(* PLC project Scenario13_Final.project, CODESYS CODESYS V3.5 SP4 Patch 4 *)
(* stored: creationDateTime 2014-06-27T19:19:34.1584235, modificationDateTime 2014-06-20T17:27:16 *)

FUNCTION_BLOCK Crane
  VAR_INPUT
    SliderNotMovedOut : BOOL;
    SliderMovedOut : BOOL;
    MagazinCapacitiveSensor : BOOL;
    WorkpieceReady : BOOL;
    CraneDown : BOOL;
    CraneUp : BOOL;
    CraneSucked : BOOL;  (* CraneOnConveyor : BOOL; CraneOnMagazin : BOOL; *)
    StampLowered : BOOL;
    MagazinOpticalSensor : BOOL;  (* CranePositionStamp : BOOL; *)
    StampSliderFilled : BOOL;
    AnalogCranePosition : INT;
    StartButtonMagazin : BOOL;
    SFCReset : BOOL;
    StartVar : BOOL;
    StampSliderSensorMovedOut : BOOL;
  END_VAR
  VAR_OUTPUT
    CraneLower : BOOL;
    MagazinVacuumOff : BOOL;
    MagazinVacuumOn : BOOL;
    CraneTurnCounterclockwise : BOOL;
    CraneTurnClockwise : BOOL;
    MagazinSlider : BOOL;
    AnalogCranePressure : INT;
    StartCommandCrane : BOOL;
  END_VAR
  VAR
    Timer1 : TON;
    Duration1 : TIME := TIME#1s500ms;
    actualtime1 : TIME;
    interconnect : BOOL;
    interconnectCraneStartCommand : BOOL;
    TimeDelay_Timer : TON;
    TimeDelay_Timer_Duration : TIME := TIME#50ms;
    TimeDelay_Timer_interconnect : BOOL;
    SFCInit : BOOL;
  END_VAR

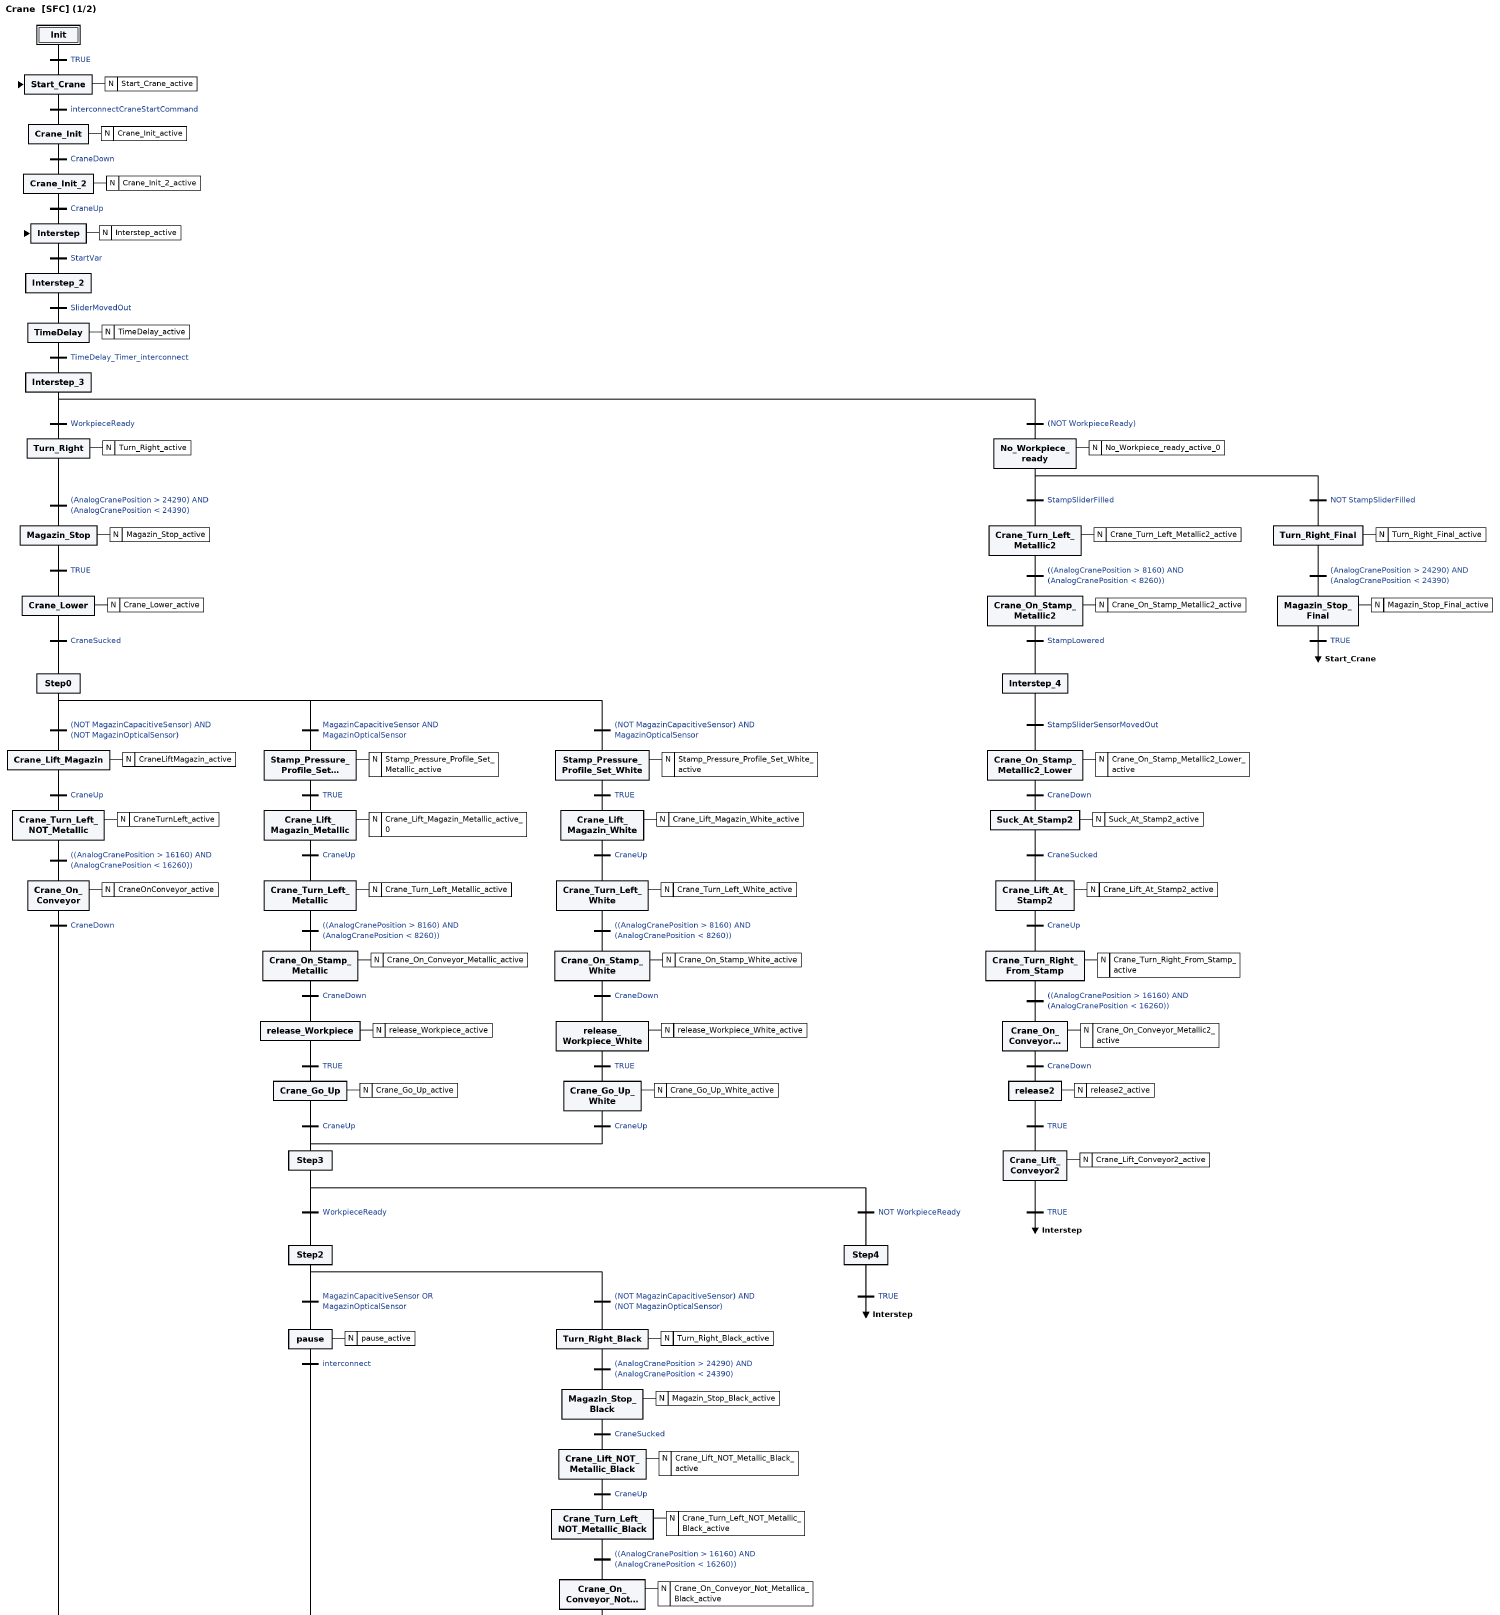
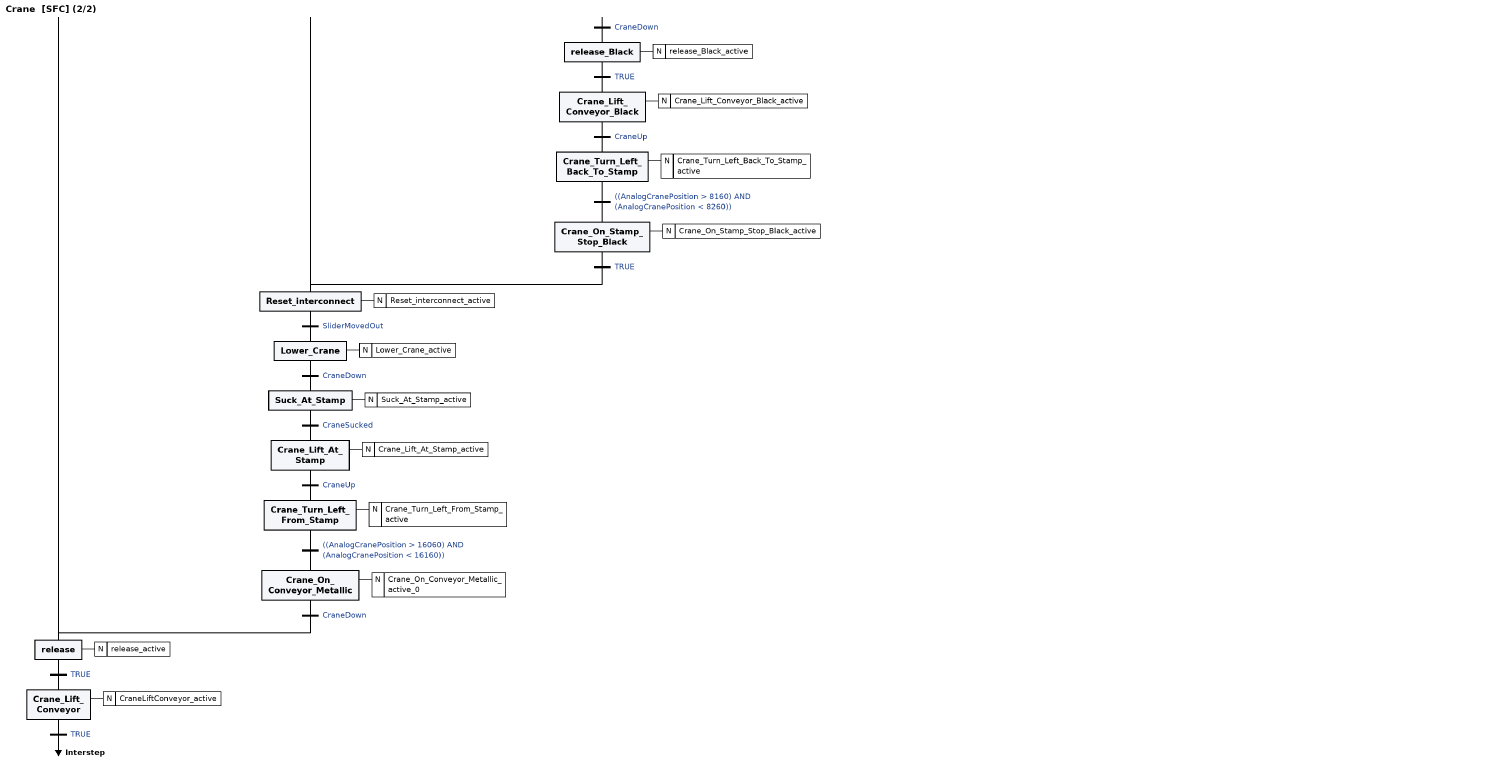
INITIAL_STEP Init:
END_STEP
TRANSITION FROM Init TO Start_Crane
  := TRUE;
END_TRANSITION
STEP Start_Crane:
  Start_Crane_active(N);
END_STEP
TRANSITION FROM Start_Crane TO Crane_Init
  := interconnectCraneStartCommand;
END_TRANSITION
STEP Crane_Init:
  Crane_Init_active(N);
END_STEP
TRANSITION FROM Crane_Init TO Crane_Init_2
  := CraneDown;
END_TRANSITION
STEP Crane_Init_2:
  Crane_Init_2_active(N);
END_STEP
TRANSITION FROM Crane_Init_2 TO Interstep
  := CraneUp;
END_TRANSITION
STEP Interstep:
  Interstep_active(N);
END_STEP
TRANSITION FROM Interstep TO Interstep_2
  := StartVar;
END_TRANSITION
STEP Interstep_2:
END_STEP
TRANSITION FROM Interstep_2 TO TimeDelay
  := SliderMovedOut;
END_TRANSITION
STEP TimeDelay:
  TimeDelay_active(N);
END_STEP
TRANSITION FROM TimeDelay TO Interstep_3
  := TimeDelay_Timer_interconnect;
END_TRANSITION
STEP Interstep_3:
END_STEP
TRANSITION FROM Interstep_3 TO Turn_Right
  := WorkpieceReady;
END_TRANSITION
TRANSITION FROM Interstep_3 TO No_Workpiece_ready
  := (NOT WorkpieceReady);
END_TRANSITION
STEP Turn_Right:
  Turn_Right_active(N);
END_STEP
TRANSITION FROM Turn_Right TO Magazin_Stop
  := (AnalogCranePosition > 24290) AND (AnalogCranePosition < 24390);
END_TRANSITION
STEP Magazin_Stop:
  Magazin_Stop_active(N);
END_STEP
TRANSITION FROM Magazin_Stop TO Crane_Lower
  := TRUE;
END_TRANSITION
STEP Crane_Lower:
  Crane_Lower_active(N);
END_STEP
TRANSITION FROM Crane_Lower TO Step0
  := CraneSucked;
END_TRANSITION
STEP Step0:
END_STEP
TRANSITION FROM Step0 TO Crane_Lift_Magazin
  := (NOT MagazinCapacitiveSensor) AND (NOT MagazinOpticalSensor);
END_TRANSITION
TRANSITION FROM Step0 TO Stamp_Pressure_Profile_Set_Metallic
  := MagazinCapacitiveSensor AND MagazinOpticalSensor;
END_TRANSITION
TRANSITION FROM Step0 TO Stamp_Pressure_Profile_Set_White
  := (NOT MagazinCapacitiveSensor) AND MagazinOpticalSensor;
END_TRANSITION
STEP Crane_Lift_Magazin:
  CraneLiftMagazin_active(N);
END_STEP
TRANSITION FROM Crane_Lift_Magazin TO Crane_Turn_Left_NOT_Metallic
  := CraneUp;
END_TRANSITION
STEP Crane_Turn_Left_NOT_Metallic:
  CraneTurnLeft_active(N);
END_STEP
TRANSITION FROM Crane_Turn_Left_NOT_Metallic TO Crane_On_Conveyor
  := ((AnalogCranePosition > 16160) AND (AnalogCranePosition < 16260));
END_TRANSITION
STEP Crane_On_Conveyor:
  CraneOnConveyor_active(N);
END_STEP
TRANSITION FROM Crane_On_Conveyor TO release
  := CraneDown;
END_TRANSITION
STEP Stamp_Pressure_Profile_Set_Metallic:
  Stamp_Pressure_Profile_Set_Metallic_active(N);
END_STEP
TRANSITION FROM Stamp_Pressure_Profile_Set_Metallic TO Crane_Lift_Magazin_Metallic
  := TRUE;
END_TRANSITION
STEP Crane_Lift_Magazin_Metallic:
  Crane_Lift_Magazin_Metallic_active_0(N);
END_STEP
TRANSITION FROM Crane_Lift_Magazin_Metallic TO Crane_Turn_Left_Metallic
  := CraneUp;
END_TRANSITION
STEP Crane_Turn_Left_Metallic:
  Crane_Turn_Left_Metallic_active(N);
END_STEP
TRANSITION FROM Crane_Turn_Left_Metallic TO Crane_On_Stamp_Metallic
  := ((AnalogCranePosition > 8160) AND (AnalogCranePosition < 8260));
END_TRANSITION
STEP Crane_On_Stamp_Metallic:
  Crane_On_Conveyor_Metallic_active(N);
END_STEP
TRANSITION FROM Crane_On_Stamp_Metallic TO release_Workpiece
  := CraneDown;
END_TRANSITION
STEP release_Workpiece:
  release_Workpiece_active(N);
END_STEP
TRANSITION FROM release_Workpiece TO Crane_Go_Up
  := TRUE;
END_TRANSITION
STEP Crane_Go_Up:
  Crane_Go_Up_active(N);
END_STEP
TRANSITION FROM Crane_Go_Up TO Step3
  := CraneUp;
END_TRANSITION
STEP Stamp_Pressure_Profile_Set_White:
  Stamp_Pressure_Profile_Set_White_active(N);
END_STEP
TRANSITION FROM Stamp_Pressure_Profile_Set_White TO Crane_Lift_Magazin_White
  := TRUE;
END_TRANSITION
STEP Crane_Lift_Magazin_White:
  Crane_Lift_Magazin_White_active(N);
END_STEP
TRANSITION FROM Crane_Lift_Magazin_White TO Crane_Turn_Left_White
  := CraneUp;
END_TRANSITION
STEP Crane_Turn_Left_White:
  Crane_Turn_Left_White_active(N);
END_STEP
TRANSITION FROM Crane_Turn_Left_White TO Crane_On_Stamp_White
  := ((AnalogCranePosition > 8160) AND (AnalogCranePosition < 8260));
END_TRANSITION
STEP Crane_On_Stamp_White:
  Crane_On_Stamp_White_active(N);
END_STEP
TRANSITION FROM Crane_On_Stamp_White TO release_Workpiece_White
  := CraneDown;
END_TRANSITION
STEP release_Workpiece_White:
  release_Workpiece_White_active(N);
END_STEP
TRANSITION FROM release_Workpiece_White TO Crane_Go_Up_White
  := TRUE;
END_TRANSITION
STEP Crane_Go_Up_White:
  Crane_Go_Up_White_active(N);
END_STEP
TRANSITION FROM Crane_Go_Up_White TO Step3
  := CraneUp;
END_TRANSITION
STEP Step3:
END_STEP
TRANSITION FROM Step3 TO Step2
  := WorkpieceReady;
END_TRANSITION
TRANSITION FROM Step3 TO Step4
  := NOT WorkpieceReady;
END_TRANSITION
STEP Step2:
END_STEP
TRANSITION FROM Step2 TO pause
  := MagazinCapacitiveSensor OR MagazinOpticalSensor;
END_TRANSITION
TRANSITION FROM Step2 TO Turn_Right_Black
  := (NOT MagazinCapacitiveSensor) AND (NOT MagazinOpticalSensor);
END_TRANSITION
STEP pause:
  pause_active(N);
END_STEP
TRANSITION FROM pause TO Reset_interconnect
  := interconnect;
END_TRANSITION
STEP Turn_Right_Black:
  Turn_Right_Black_active(N);
END_STEP
TRANSITION FROM Turn_Right_Black TO Magazin_Stop_Black
  := (AnalogCranePosition > 24290) AND (AnalogCranePosition < 24390);
END_TRANSITION
STEP Magazin_Stop_Black:
  Magazin_Stop_Black_active(N);
END_STEP
TRANSITION FROM Magazin_Stop_Black TO Crane_Lift_NOT_Metallic_Black
  := CraneSucked;
END_TRANSITION
STEP Crane_Lift_NOT_Metallic_Black:
  Crane_Lift_NOT_Metallic_Black_active(N);
END_STEP
TRANSITION FROM Crane_Lift_NOT_Metallic_Black TO Crane_Turn_Left_NOT_Metallic_Black
  := CraneUp;
END_TRANSITION
STEP Crane_Turn_Left_NOT_Metallic_Black:
  Crane_Turn_Left_NOT_Metallic_Black_active(N);
END_STEP
TRANSITION FROM Crane_Turn_Left_NOT_Metallic_Black TO Crane_On_Conveyor_Not_Metallica_Black
  := ((AnalogCranePosition > 16160) AND (AnalogCranePosition < 16260));
END_TRANSITION
STEP Crane_On_Conveyor_Not_Metallica_Black:
  Crane_On_Conveyor_Not_Metallica_Black_active(N);
END_STEP
TRANSITION FROM Crane_On_Conveyor_Not_Metallica_Black TO release_Black
  := CraneDown;
END_TRANSITION
STEP release_Black:
  release_Black_active(N);
END_STEP
TRANSITION FROM release_Black TO Crane_Lift_Conveyor_Black
  := TRUE;
END_TRANSITION
STEP Crane_Lift_Conveyor_Black:
  Crane_Lift_Conveyor_Black_active(N);
END_STEP
TRANSITION FROM Crane_Lift_Conveyor_Black TO Crane_Turn_Left_Back_To_Stamp
  := CraneUp;
END_TRANSITION
STEP Crane_Turn_Left_Back_To_Stamp:
  Crane_Turn_Left_Back_To_Stamp_active(N);
END_STEP
TRANSITION FROM Crane_Turn_Left_Back_To_Stamp TO Crane_On_Stamp_Stop_Black
  := ((AnalogCranePosition > 8160) AND (AnalogCranePosition < 8260));
END_TRANSITION
STEP Crane_On_Stamp_Stop_Black:
  Crane_On_Stamp_Stop_Black_active(N);
END_STEP
TRANSITION FROM Crane_On_Stamp_Stop_Black TO Reset_interconnect
  := TRUE;
END_TRANSITION
STEP Step4:
END_STEP
TRANSITION FROM Step4 TO Interstep
  := TRUE;
END_TRANSITION
STEP Reset_interconnect:
  Reset_interconnect_active(N);
END_STEP
TRANSITION FROM Reset_interconnect TO Lower_Crane
  := SliderMovedOut;
END_TRANSITION
STEP Lower_Crane:
  Lower_Crane_active(N);
END_STEP
TRANSITION FROM Lower_Crane TO Suck_At_Stamp
  := CraneDown;
END_TRANSITION
STEP Suck_At_Stamp:
  Suck_At_Stamp_active(N);
END_STEP
TRANSITION FROM Suck_At_Stamp TO Crane_Lift_At_Stamp
  := CraneSucked;
END_TRANSITION
STEP Crane_Lift_At_Stamp:
  Crane_Lift_At_Stamp_active(N);
END_STEP
TRANSITION FROM Crane_Lift_At_Stamp TO Crane_Turn_Left_From_Stamp
  := CraneUp;
END_TRANSITION
STEP Crane_Turn_Left_From_Stamp:
  Crane_Turn_Left_From_Stamp_active(N);
END_STEP
TRANSITION FROM Crane_Turn_Left_From_Stamp TO Crane_On_Conveyor_Metallic
  := ((AnalogCranePosition > 16060) AND (AnalogCranePosition < 16160));
END_TRANSITION
STEP Crane_On_Conveyor_Metallic:
  Crane_On_Conveyor_Metallic_active_0(N);
END_STEP
TRANSITION FROM Crane_On_Conveyor_Metallic TO release
  := CraneDown;
END_TRANSITION
STEP release:
  release_active(N);
END_STEP
TRANSITION FROM release TO Crane_Lift_Conveyor
  := TRUE;
END_TRANSITION
STEP Crane_Lift_Conveyor:
  CraneLiftConveyor_active(N);
END_STEP
TRANSITION FROM Crane_Lift_Conveyor TO Interstep
  := TRUE;
END_TRANSITION
STEP No_Workpiece_ready:
  No_Workpiece_ready_active_0(N);
END_STEP
TRANSITION FROM No_Workpiece_ready TO Crane_Turn_Left_Metallic2
  := StampSliderFilled;
END_TRANSITION
TRANSITION FROM No_Workpiece_ready TO Turn_Right_Final
  := NOT StampSliderFilled;
END_TRANSITION
STEP Crane_Turn_Left_Metallic2:
  Crane_Turn_Left_Metallic2_active(N);
END_STEP
TRANSITION FROM Crane_Turn_Left_Metallic2 TO Crane_On_Stamp_Metallic2
  := ((AnalogCranePosition > 8160) AND (AnalogCranePosition < 8260));
END_TRANSITION
STEP Crane_On_Stamp_Metallic2:
  Crane_On_Stamp_Metallic2_active(N);
END_STEP
TRANSITION FROM Crane_On_Stamp_Metallic2 TO Interstep_4
  := StampLowered;
END_TRANSITION
STEP Interstep_4:
END_STEP
TRANSITION FROM Interstep_4 TO Crane_On_Stamp_Metallic2_Lower
  := StampSliderSensorMovedOut;
END_TRANSITION
STEP Crane_On_Stamp_Metallic2_Lower:
  Crane_On_Stamp_Metallic2_Lower_active(N);
END_STEP
TRANSITION FROM Crane_On_Stamp_Metallic2_Lower TO Suck_At_Stamp2
  := CraneDown;
END_TRANSITION
STEP Suck_At_Stamp2:
  Suck_At_Stamp2_active(N);
END_STEP
TRANSITION FROM Suck_At_Stamp2 TO Crane_Lift_At_Stamp2
  := CraneSucked;
END_TRANSITION
STEP Crane_Lift_At_Stamp2:
  Crane_Lift_At_Stamp2_active(N);
END_STEP
TRANSITION FROM Crane_Lift_At_Stamp2 TO Crane_Turn_Right_From_Stamp
  := CraneUp;
END_TRANSITION
STEP Crane_Turn_Right_From_Stamp:
  Crane_Turn_Right_From_Stamp_active(N);
END_STEP
TRANSITION FROM Crane_Turn_Right_From_Stamp TO Crane_On_Conveyor_Metallic2
  := ((AnalogCranePosition > 16160) AND (AnalogCranePosition < 16260));
END_TRANSITION
STEP Crane_On_Conveyor_Metallic2:
  Crane_On_Conveyor_Metallic2_active(N);
END_STEP
TRANSITION FROM Crane_On_Conveyor_Metallic2 TO release2
  := CraneDown;
END_TRANSITION
STEP release2:
  release2_active(N);
END_STEP
TRANSITION FROM release2 TO Crane_Lift_Conveyor2
  := TRUE;
END_TRANSITION
STEP Crane_Lift_Conveyor2:
  Crane_Lift_Conveyor2_active(N);
END_STEP
TRANSITION FROM Crane_Lift_Conveyor2 TO Interstep
  := TRUE;
END_TRANSITION
STEP Turn_Right_Final:
  Turn_Right_Final_active(N);
END_STEP
TRANSITION FROM Turn_Right_Final TO Magazin_Stop_Final
  := (AnalogCranePosition > 24290) AND (AnalogCranePosition < 24390);
END_TRANSITION
STEP Magazin_Stop_Final:
  Magazin_Stop_Final_active(N);
END_STEP
TRANSITION FROM Magazin_Stop_Final TO Start_Crane
  := TRUE;
END_TRANSITION

ACTION Turn_Right_Final_active:
                CraneTurnClockwise := TRUE;
CraneTurnCounterclockwise := FALSE;
AnalogCranePressure := 0;
              
END_ACTION

ACTION Crane_Turn_Right_From_Stamp_active:
                CraneTurnClockwise := TRUE;
CraneTurnCounterclockwise := FALSE;
              
END_ACTION

ACTION Crane_On_Stamp_Metallic2_active:
                CraneTurnCounterclockwise := FALSE;
CraneTurnClockwise := FALSE;
              
END_ACTION

ACTION Crane_Turn_Left_White_active:
                CraneTurnCounterclockwise := TRUE;
CraneTurnClockwise := FALSE;
              
END_ACTION

ACTION Suck_At_Stamp_active:
                MagazinVacuumOn := TRUE;
MagazinVacuumOff := FALSE;
              
END_ACTION

ACTION release_Black_active:
                MagazinVacuumOn := FALSE;
MagazinVacuumOff := TRUE;
              
END_ACTION

ACTION Crane_Lift_Magazin_Metallic_active_0:
                CraneLower := FALSE;
              
END_ACTION

ACTION Reset_interconnect_active:
                interconnect := FALSE;
Timer1(IN:=FALSE,PT:=T#1ms);
              
END_ACTION

ACTION CraneOnConveyor_active:
                CraneTurnCounterclockwise := FALSE;
CraneTurnClockwise := FALSE;
CraneLower := TRUE;
              
END_ACTION

ACTION Crane_Go_Up_White_active:
                CraneLower := FALSE;
              
END_ACTION

ACTION Crane_On_Conveyor_Metallic_active:
                CraneTurnCounterclockwise := FALSE;
CraneTurnClockwise := FALSE;
CraneLower := TRUE;
              
END_ACTION

ACTION Crane_Turn_Left_Metallic_active:
                CraneTurnCounterclockwise := TRUE;
CraneTurnClockwise := FALSE;
              
END_ACTION

ACTION CraneLiftMagazin_active:
                CraneLower := FALSE;
              
END_ACTION

ACTION release2_active:
                MagazinVacuumOff := TRUE;
MagazinVacuumOn := FALSE;
              
END_ACTION

ACTION Crane_Turn_Left_Metallic2_active:
                CraneTurnCounterclockwise := TRUE;
CraneTurnClockwise := FALSE;
              
END_ACTION

ACTION Magazin_Stop_Final_active:
                CraneTurnClockwise := FALSE;
CraneTurnCounterClockwise := FALSE;
              
END_ACTION

ACTION Interstep_active:
                StartCommandCrane := TRUE;
              
END_ACTION

ACTION Magazin_Stop_active:
                CraneTurnClockwise := FALSE;
CraneTurnCounterClockwise := FALSE;
              
END_ACTION

ACTION Lower_Crane_active:
                CraneLower := TRUE;
              
END_ACTION

ACTION Crane_Lift_Magazin_White_active:
                CraneLower := FALSE;
              
END_ACTION

ACTION release_Workpiece_White_active:
                MagazinVacuumOff := TRUE;
MagazinVacuumOn := FALSE;
              
END_ACTION

ACTION Crane_On_Stamp_White_active:
                CraneTurnCounterclockwise := FALSE;
CraneTurnClockwise := FALSE;
CraneLower := TRUE;
              
END_ACTION

ACTION release_Workpiece_active:
                MagazinVacuumOff := TRUE;
MagazinVacuumOn := FALSE;
              
END_ACTION

ACTION No_Workpiece_ready_active_0:
                MagazinVacuumOn := FALSE;
MagazinVacuumOff := FALSE;
CraneLower := FALSE;

              
END_ACTION

ACTION Crane_Turn_Left_Back_To_Stamp_active:
                CraneTurnCounterclockwise := TRUE;
CraneTurnClockwise := FALSE;
              
END_ACTION

ACTION Crane_Lift_Conveyor_Black_active:
                CraneLower := FALSE;
              
END_ACTION

ACTION Crane_Lift_At_Stamp_active:
                CraneLower := FALSE;
              
END_ACTION

ACTION Crane_Lift_At_Stamp2_active:
                CraneLower := FALSE;
AnalogCranePressure := 0;
              
END_ACTION

ACTION Crane_On_Conveyor_Not_Metallica_Black_active:
                CraneTurnCounterclockwise := FALSE;
CraneTurnClockwise := FALSE;
CraneLower := TRUE;
              
END_ACTION

ACTION Crane_Lift_Conveyor2_active:
                CraneLower := FALSE;
              
END_ACTION

ACTION Crane_Init_2_active:
                CraneLower := FALSE;
              
END_ACTION

ACTION Start_Crane_active:
                CraneLower := FALSE;
MagazinVacuumOff := FALSE;
MagazinVacuumOn := FALSE;
CraneTurnCounterclockwise := FALSE;
CraneTurnClockwise := FALSE;
AnalogCranePressure := 0;
StartVar := FALSE;
StartCommandCrane := FALSE;


IF(StartButtonMagazin = TRUE) THEN
	interconnectCraneStartCommand := TRUE;
END_IF
              
END_ACTION

ACTION Suck_At_Stamp2_active:
                MagazinVacuumOn := TRUE;
MagazinVacuumOff := FALSE;
              
END_ACTION

ACTION Stamp_Pressure_Profile_Set_White_active:
                AnalogCranePressure := 6000;
              
END_ACTION

ACTION Turn_Right_Black_active:
                CraneTurnClockwise := TRUE;
CraneTurnCounterclockwise := FALSE;
              
END_ACTION

ACTION release_active:
                MagazinVacuumOff := TRUE;
MagazinVacuumOn := FALSE;
              
END_ACTION

ACTION Crane_Lower_active:
                MagazinVacuumOn := TRUE;
MagazinVacuumOff := FALSE;
CraneLower := TRUE;
AnalogCranePressure := 0;
              
END_ACTION

ACTION Crane_On_Stamp_Stop_Black_active:
                CraneTurnClockwise := FALSE;
CraneTurnCounterclockwise := FALSE;
              
END_ACTION

ACTION Stamp_Pressure_Profile_Set_Metallic_active:
                AnalogCranePressure := 7000;
              
END_ACTION

ACTION Crane_On_Conveyor_Metallic_active_0:
                CraneTurnCounterclockwise := FALSE;
CraneTurnClockwise := FALSE;
CraneLower := TRUE;
              
END_ACTION

ACTION Turn_Right_active:
                CraneTurnClockwise := TRUE;
CraneTurnCounterclockwise := FALSE;
              
END_ACTION

ACTION pause_active:
                Timer1(IN:=CraneUP, PT:=Duration1);
interconnect := Timer1.Q;
              
END_ACTION

ACTION TimeDelay_active:
                TimeDelay_Timer(IN:=TRUE, PT:=TimeDelay_Timer_Duration);
TimeDelay_Timer_interconnect := TimeDelay_Timer.Q;
              
END_ACTION

ACTION Crane_Init_active:
                CraneLower := TRUE;
interconnectCraneStartCommand := FALSE;
AnalogCranePressure := 6000;
              
END_ACTION

ACTION Crane_Go_Up_active:
                CraneLower := FALSE;
              
END_ACTION

ACTION CraneTurnLeft_active:
                CraneTurnCounterclockwise := TRUE;
CraneTurnClockwise := FALSE;
              
END_ACTION

ACTION Magazin_Stop_Black_active:
                CraneTurnClockwise := FALSE;
CraneTurnCounterclockwise := FALSE;
MagazinVacuumOn := TRUE;
MagazinVacuumOff := FALSE;
CraneLower := TRUE;
              
END_ACTION

ACTION Crane_On_Stamp_Metallic2_Lower_active:
                CraneLower := TRUE;
              
END_ACTION

ACTION CraneLiftConveyor_active:
                CraneLower := FALSE;
              
END_ACTION

ACTION Crane_Turn_Left_NOT_Metallic_Black_active:
                CraneTurnCounterclockwise := TRUE;
CraneTurnClockwise := FALSE;
              
END_ACTION

ACTION Crane_Turn_Left_From_Stamp_active:
                CraneTurnClockwise := TRUE;
CraneTurnCounterclockwise := FALSE;
              
END_ACTION

ACTION Crane_On_Conveyor_Metallic2_active:
                CraneTurnCounterclockwise := FALSE;
CraneTurnClockwise := FALSE;
CraneLower := TRUE;
              
END_ACTION

ACTION Crane_Lift_NOT_Metallic_Black_active:
                CraneLower := FALSE;
              
END_ACTION
END_FUNCTION_BLOCK

FUNCTION_BLOCK Magazin
  VAR_INPUT
    SliderNotMovedOut : BOOL;
    SliderMovedOut : BOOL;
    WorkpieceReady : BOOL;
    CraneDown : BOOL;
    CraneUp : BOOL;
    CraneOnConveyor : BOOL;
    CraneOnMagazin : BOOL;
    CraneSucked : BOOL;
    AnalogCranePosition : INT;
    StartButtonMagazin : BOOL;
    SFCReset : BOOL;
    StartVar : BOOL;
  END_VAR
  VAR_OUTPUT
    CraneLower : BOOL;
    MagazinVacuumOff : BOOL;
    MagazinVacuumOn : BOOL;
    CraneTurnCounterclockwise : BOOL;
    CraneTurnClockwise : BOOL;
    MagazinSlider : BOOL;
    MagazinGreenLamp : BOOL;
    MagazinWhiteLamp : BOOL;
    StartCommandMagazin : BOOL;
  END_VAR
  VAR
    interconnectMagazinStartCommand : BOOL;
    SFCInit : BOOL;
  END_VAR

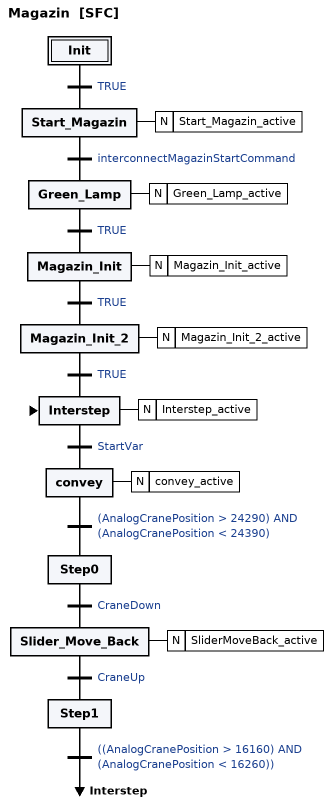
INITIAL_STEP Init:
END_STEP
TRANSITION FROM Init TO Start_Magazin
  := TRUE;
END_TRANSITION
STEP Start_Magazin:
  Start_Magazin_active(N);
END_STEP
TRANSITION FROM Start_Magazin TO Green_Lamp
  := interconnectMagazinStartCommand;
END_TRANSITION
STEP Green_Lamp:
  Green_Lamp_active(N);
END_STEP
TRANSITION FROM Green_Lamp TO Magazin_Init
  := TRUE;
END_TRANSITION
STEP Magazin_Init:
  Magazin_Init_active(N);
END_STEP
TRANSITION FROM Magazin_Init TO Magazin_Init_2
  := TRUE;
END_TRANSITION
STEP Magazin_Init_2:
  Magazin_Init_2_active(N);
END_STEP
TRANSITION FROM Magazin_Init_2 TO Interstep
  := TRUE;
END_TRANSITION
STEP Interstep:
  Interstep_active(N);
END_STEP
TRANSITION FROM Interstep TO convey
  := StartVar;
END_TRANSITION
STEP convey:
  convey_active(N);
END_STEP
TRANSITION FROM convey TO Step0
  := (AnalogCranePosition > 24290) AND (AnalogCranePosition < 24390);
END_TRANSITION
STEP Step0:
END_STEP
TRANSITION FROM Step0 TO Slider_Move_Back
  := CraneDown;
END_TRANSITION
STEP Slider_Move_Back:
  SliderMoveBack_active(N);
END_STEP
TRANSITION FROM Slider_Move_Back TO Step1
  := CraneUp;
END_TRANSITION
STEP Step1:
END_STEP
TRANSITION FROM Step1 TO Interstep
  := ((AnalogCranePosition > 16160) AND (AnalogCranePosition < 16260));
END_TRANSITION

ACTION Start_Magazin_active:
                MagazinSlider := FALSE;
MagazinGreenLamp := FALSE;
StartVar := FALSE;
StartCommandMagazin := FALSE;


IF(StartButtonMagazin = TRUE) THEN
	interconnectMagazinStartCommand := TRUE;
END_IF
              
END_ACTION

ACTION Magazin_Init_active:
                MagazinSlider := TRUE;
              
END_ACTION

ACTION Interstep_active:
                StartCommandMagazin := TRUE;
              
END_ACTION

ACTION SliderMoveBack_active:
                IF((SliderMovedOut = TRUE)AND(SliderNotMovedOut = FALSE))THEN
	MagazinSlider := FALSE;
END_IF
              
END_ACTION

ACTION Magazin_Init_2_active:
                MagazinSlider := FALSE;
              
END_ACTION

ACTION convey_active:
                IF(SliderNotMovedOut)THEN
	MagazinSlider := TRUE;
END_IF
              
END_ACTION

ACTION Green_Lamp_active:
                MagazinGreenLamp := TRUE;
interconnectMagazinStartCommand := FALSE;
              
END_ACTION
END_FUNCTION_BLOCK

FUNCTION_BLOCK Conveyor
  VAR_INPUT
    SorterStartButton : BOOL;
    SorterSwitchManuellAutomatic : BOOL;
    SorterLightbarrierCraneInterface : BOOL;
    SFCReset : BOOL;
    StartVar : BOOL;
  END_VAR
  VAR_OUTPUT
    SorterConveyorTowardsStacker : BOOL;
    SorterConveyorTowardsCrane : BOOL;
    SorterGreenLampConveyor : BOOL;
    SorterWhiteLampConveyor : BOOL;
    StartCommandConveyor : BOOL;
  END_VAR
  VAR
    interconnectConveyorStartCommand : BOOL;
    interconnectConveyorTerminationCommand : BOOL;
    Timer_Conveyor_Runtime : TON;
    Duration_Conveyor_Runtime : TIME := TIME#4s500ms;
    interconnect_Conveyor_Runtime : BOOL;
    Timer_Conveyor_Test : TON;
    Duration_Conveyor_Test : TIME := TIME#1s0ms;
    interconnect_Conveyor_Test : BOOL;
    SFCInit : BOOL;
  END_VAR

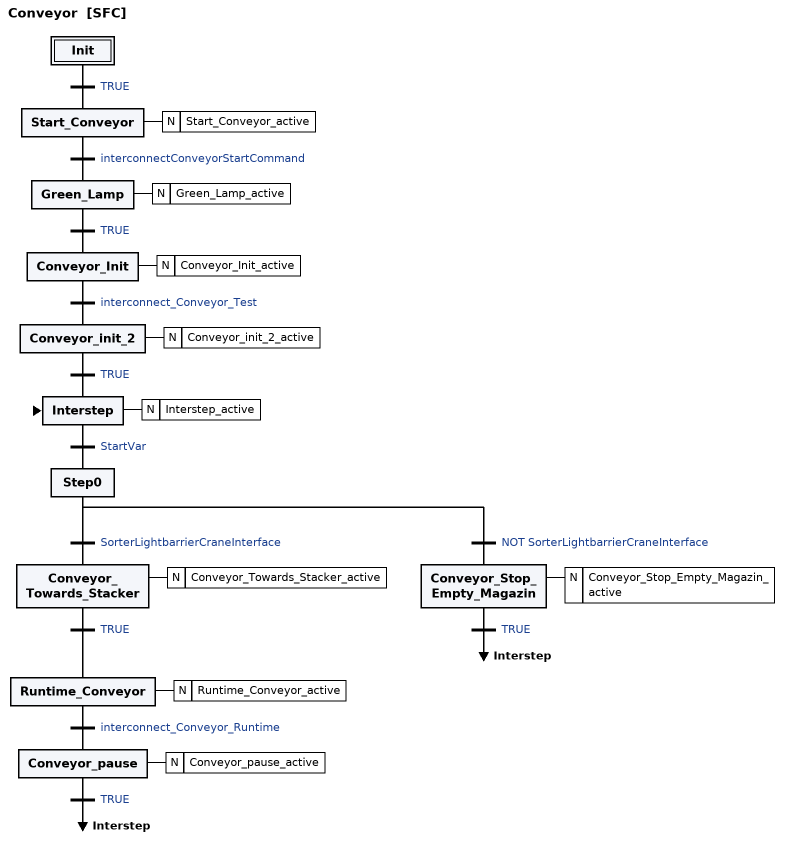
INITIAL_STEP Init:
END_STEP
TRANSITION FROM Init TO Start_Conveyor
  := TRUE;
END_TRANSITION
STEP Start_Conveyor:
  Start_Conveyor_active(N);
END_STEP
TRANSITION FROM Start_Conveyor TO Green_Lamp
  := interconnectConveyorStartCommand;
END_TRANSITION
STEP Green_Lamp:
  Green_Lamp_active(N);
END_STEP
TRANSITION FROM Green_Lamp TO Conveyor_Init
  := TRUE;
END_TRANSITION
STEP Conveyor_Init:
  Conveyor_Init_active(N);
END_STEP
TRANSITION FROM Conveyor_Init TO Conveyor_init_2
  := interconnect_Conveyor_Test;
END_TRANSITION
STEP Conveyor_init_2:
  Conveyor_init_2_active(N);
END_STEP
TRANSITION FROM Conveyor_init_2 TO Interstep
  := TRUE;
END_TRANSITION
STEP Interstep:
  Interstep_active(N);
END_STEP
TRANSITION FROM Interstep TO Step0
  := StartVar;
END_TRANSITION
STEP Step0:
END_STEP
TRANSITION FROM Step0 TO Conveyor_Towards_Stacker
  := SorterLightbarrierCraneInterface;
END_TRANSITION
TRANSITION FROM Step0 TO Conveyor_Stop_Empty_Magazin
  := NOT SorterLightbarrierCraneInterface;
END_TRANSITION
STEP Conveyor_Towards_Stacker:
  Conveyor_Towards_Stacker_active(N);
END_STEP
TRANSITION FROM Conveyor_Towards_Stacker TO Runtime_Conveyor
  := TRUE;
END_TRANSITION
STEP Runtime_Conveyor:
  Runtime_Conveyor_active(N);
END_STEP
TRANSITION FROM Runtime_Conveyor TO Conveyor_pause
  := interconnect_Conveyor_Runtime;
END_TRANSITION
STEP Conveyor_pause:
  Conveyor_pause_active(N);
END_STEP
TRANSITION FROM Conveyor_pause TO Interstep
  := TRUE;
END_TRANSITION
STEP Conveyor_Stop_Empty_Magazin:
  Conveyor_Stop_Empty_Magazin_active(N);
END_STEP
TRANSITION FROM Conveyor_Stop_Empty_Magazin TO Interstep
  := TRUE;
END_TRANSITION

ACTION Conveyor_pause_active:
                SorterConveyorTowardsStacker := FALSE;
SorterConveyorTowardsCrane := FALSE;
interconnect_Conveyor_Runtime := FALSE;
Timer_Conveyor_Runtime(IN:=FALSE,PT:=T#0MS);
              
END_ACTION

ACTION Conveyor_init_2_active:
                SorterConveyorTowardsStacker := FALSE;
SorterConveyorTowardsCrane := FALSE;
interconnect_Conveyor_Test := FALSE;
Timer_Conveyor_Test(IN:=FALSE,PT:=T#0MS);
              
END_ACTION

ACTION Start_Conveyor_active:
                interconnectConveyorTerminationCommand := FALSE;
SorterConveyorTowardsStacker := FALSE;
SorterConveyorTowardsCrane := FALSE;
SorterGreenLampConveyor := FALSE;
interconnect_Conveyor_Runtime := FALSE;
interconnect_Conveyor_Test := FALSE;
Timer_Conveyor_Test(IN:=FALSE,PT:=T#0MS);
Timer_Conveyor_Runtime(IN:=FALSE,PT:=T#0MS);
StartVar := FALSE;
StartCommandConveyor := FALSE;

IF(SorterStartButton = TRUE) THEN
	interconnectConveyorStartCommand := TRUE;
END_IF
              
END_ACTION

ACTION Green_Lamp_active:
                SorterGreenLampConveyor := TRUE;
interconnectConveyorStartCommand := FALSE;
              
END_ACTION

ACTION Runtime_Conveyor_active:
                Timer_Conveyor_Runtime(IN:=TRUE, PT:=Duration_Conveyor_Runtime);
interconnect_Conveyor_Runtime := Timer_Conveyor_Runtime.Q;
              
END_ACTION

ACTION Conveyor_Stop_Empty_Magazin_active:
                SorterConveyorTowardsStacker := FALSE;
SorterConveyorTowardsCrane := FALSE;
interconnectConveyorStartCommand := FALSE;
              
END_ACTION

ACTION Conveyor_Stop_active:
                SorterConveyorTowardsStacker := FALSE;
SorterConveyorTowardsCrane := FALSE;
SorterGreenLampConveyor := FALSE;
interconnectConveyorStartCommand := FALSE;
              
END_ACTION

ACTION Conveyor_Init_active:
                SorterConveyorTowardsStacker := TRUE;
SorterConveyorTowardsCrane := FALSE;
Timer_Conveyor_Test(IN:=TRUE, PT:=Duration_Conveyor_Test);
interconnect_Conveyor_Test := Timer_Conveyor_Test.Q;
              
END_ACTION

ACTION Conveyor_Towards_Stacker_active:
                SorterConveyorTowardsStacker := TRUE;
SorterConveyorTowardsCrane := FALSE;
              
END_ACTION

ACTION Interstep_active:
                StartCommandConveyor := TRUE;
              
END_ACTION
END_FUNCTION_BLOCK

PROGRAM Main
  VAR
    Sensor_StartButtonMagazin : BOOL;
    Sensor_MagazinEmergencyStop : BOOL;
    Sensor_MagazinSwitchManuellAutomatic : BOOL;
    Sensor_CraneSucked : BOOL;
    Sensor_CraneDown : BOOL;
    Sensor_CraneUp : BOOL;
    Sensor_SliderNotMovedOut : BOOL;
    Sensor_SliderMovedOut : BOOL;
    Sensor_MagazinCapacitiveSensor : BOOL;
    Sensor_MagazinOpticalSensor : BOOL;
    Sensor_CranePositionStamp : BOOL;
    Sensor_CraneOnConveyor : BOOL;
    Sensor_CraneOnMagazin : BOOL;
    Sensor_WorkpieceReady : BOOL;
    Sensor_CranePosition : BOOL;
    Sensor_StampSliderSensorMovedOut : BOOL;
    Sensor_StampSliderSensorMovedIn : BOOL;
    Sensor_StampSliderFilled : BOOL;
    Sensor_StampUp : BOOL;
    Sensor_StampLowered : BOOL;
    Sensor_StampSwitchManuellAutomatic : BOOL;
    Sensor_StampEmergencyStop : BOOL;
    Sensor_StampStartButton : BOOL;
    Sensor_SorterLightnesssensorCraneInterfaceInverse : BOOL;
    Sensor_SorterLightbarrierCraneInterface : BOOL;
    Sensor_SorterCapacitiveSensorPusher1 : BOOL;
    Sensor_SorterLightnessSensorPusher1 : BOOL;
    Sensor_SorterCapacitiveSensorPusher2 : BOOL;
    Sensor_SorterLightnessSensorPusher2 : BOOL;
    Sensor_SorterLightnessSensorPusher3 : BOOL;
    Sensor_SorterPusher1MovedOut : BOOL;
    Sensor_SorterPusher1MovedIn : BOOL;
    Sensor_SorterPusher2MovedOut : BOOL;
    Sensor_SorterPusher2MovedIn : BOOL;
    Sensor_SorterEmergencyStop : BOOL;
    Sensor_SorterStartButton : BOOL;
    Sensor_SorterSwitchManuellAutomatic : BOOL;
    Sensor_AnalogCranePosition : INT;  (* Max: 27449 // Min: 5070 // Stempel: 8120 // Magazin: 24340 // Laufband: 16270 *)
    Actuator_MagazinSlider : BOOL;
    Actuator_CraneLower : BOOL;
    Actuator_MagazinVacuumOn : BOOL;
    Actuator_MagazinVacuumOff : BOOL;
    Actuator_MagazinGreenLamp : BOOL;
    Actuator_MagazinWhiteLamp : BOOL;
    Actuator_CraneTurnCounterclockwise : BOOL;
    Actuator_CraneTurnClockwise : BOOL;
    Actuator_SorterConveyorTowardsStacker : BOOL;
    Actuator_SorterConveyorTowardsCrane : BOOL;
    Actuator_SorterGreenLampConveyor : BOOL;
    Actuator_SorterWhiteLampConveyor : BOOL;
    Actuator_PusherY1 : BOOL;
    Actuator_PusherY2 : BOOL;
    Actuator_StampSliderMovedOut : BOOL;
    Actuator_StampSliderMovedIn : BOOL;
    Actuator_StampWhiteLamp : BOOL;
    Actuator_StampGreenLamp : BOOL;
    Actuator_StampPusher : BOOL;
    Actuator_AnalogCranePressure : INT;
    Mag : Magazin;
    Crane : Crane;
    Stamp : Stamp;
    Conveyor : Conveyor;
    Pusher : Pusher;
  END_VAR

            Mag.SliderNotMovedOut := Sensor_SliderNotMovedOut;
Mag.SliderMovedOut := Sensor_SliderMovedOut;
Mag.CraneOnMagazin := Sensor_CraneOnMagazin;
Mag.CraneDown := Sensor_CraneDown;
Mag.CraneUp := Sensor_CraneUp;
Mag.CraneOnConveyor := Sensor_CraneOnConveyor;
Mag.WorkpieceReady := Sensor_WorkpieceReady;
Mag.AnalogCranePosition := Sensor_AnalogCranePosition;
Mag.StartButtonMagazin := Sensor_StartButtonMagazin;

Actuator_MagazinSlider := Mag.MagazinSlider;
Actuator_MagazinGreenLamp := Mag.MagazinGreenLamp;


Crane.CraneUp := Sensor_CraneUp;
(*Crane.CraneOnConveyor := Sensor_CraneOnConveyor;*)
Crane.CraneDown := Sensor_CraneDown;
Crane.CraneSucked := Sensor_CraneSucked;
(*Crane.CraneOnMagazin := Sensor_CraneOnMagazin;*)
Crane.MagazinCapacitiveSensor := Sensor_MagazinCapacitiveSensor;
(*Crane.CranePositionStamp := Sensor_CranePositionStamp;*)
Crane.SliderMovedOut := Sensor_SliderMovedOut;
Crane.WorkpieceReady := Sensor_WorkpieceReady;
Crane.MagazinOpticalSensor := Sensor_MagazinOpticalSensor;
Crane.StampSliderFilled := Sensor_StampSliderFilled;
Crane.StampSliderSensorMovedOut := Sensor_StampSliderSensorMovedOut;
Crane.StampLowered := Sensor_StampLowered;
Crane.AnalogCranePosition := Sensor_AnalogCranePosition;
Crane.StartButtonMagazin := Sensor_StartButtonMagazin;

Actuator_CraneTurnCounterclockwise := Crane.CraneTurnCounterclockwise;
Actuator_CraneTurnClockwise := Crane.CraneTurnClockwise;
Actuator_CraneLower := Crane.CraneLower;
Actuator_MagazinVacuumOff := Crane.MagazinVacuumOff;
Actuator_MagazinVacuumOn := Crane.MagazinVacuumOn;
Actuator_AnalogCranePressure := Crane.AnalogCranePressure;



Stamp.StampSliderSensorMovedOut := Sensor_StampSliderSensorMovedOut;
Stamp.StampSliderSensorMovedIn := Sensor_StampSliderSensorMovedIn;
Stamp.StampSliderFilled := Sensor_StampSliderFilled;
Stamp.StampUp := Sensor_StampUp;
Stamp.StampLowered := Sensor_StampLowered;
Stamp.CraneDown := Sensor_CraneDown;
Stamp.CraneUp := Sensor_CraneUp;
Stamp.CraneSucked := Sensor_CraneSucked;
Stamp.CranePositionStamp := Sensor_CranePositionStamp;
Stamp.CraneOnConveyor := Sensor_CraneOnConveyor;
Stamp.AnalogCranePosition := Sensor_AnalogCranePosition;
Stamp.StampStartButton := Sensor_StampStartButton;

Actuator_StampSliderMovedOut := Stamp.StampSliderMovedOut;
Actuator_StampSliderMovedIn := Stamp.StampSliderMovedIn;
Actuator_StampWhiteLamp := Stamp.StampWhiteLamp;
Actuator_StampPusher := Stamp.StampPusher;
Actuator_StampGreenLamp := Stamp.StampGreenLamp;


Conveyor.SorterStartButton := Sensor_SorterStartButton;
Conveyor.SorterSwitchManuellAutomatic := Sensor_SorterSwitchManuellAutomatic;
Conveyor.SorterLightbarrierCraneInterface := Sensor_SorterLightbarrierCraneInterface;

Actuator_SorterConveyorTowardsStacker := Conveyor.SorterConveyorTowardsStacker;
Actuator_SorterConveyorTowardsCrane := Conveyor.SorterConveyorTowardsCrane;
Actuator_SorterGreenLampConveyor := Conveyor.SorterGreenLampConveyor;
Actuator_SorterWhiteLampConveyor := Conveyor.SorterWhiteLampConveyor;


Pusher.SorterLightnesssensorCraneInterfaceInverse := Sensor_SorterLightnesssensorCraneInterfaceInverse;
Pusher.SorterLightbarrierCraneInterface := Sensor_SorterLightbarrierCraneInterface;
Pusher.SorterCapacitiveSensorPusher1 := Sensor_SorterCapacitiveSensorPusher1;
Pusher.SorterLightnessSensorPusher1 := Sensor_SorterLightnessSensorPusher1;
Pusher.SorterCapacitiveSensorPusher2 :=	Sensor_SorterCapacitiveSensorPusher2;
Pusher.SorterLightnessSensorPusher2 := Sensor_SorterLightnessSensorPusher2;
Pusher.SorterLightnessSensorPusher3 := Sensor_SorterLightnessSensorPusher3;
Pusher.SorterPusher1MovedOut := Sensor_SorterPusher1MovedOut;
Pusher.SorterPusher1MovedIn := Sensor_SorterPusher1MovedIn;
Pusher.SorterPusher2MovedOut := Sensor_SorterPusher2MovedOut;
Pusher.SorterPusher2MovedIn := Sensor_SorterPusher2MovedIn;
Pusher.SorterStartButton := Sensor_SorterStartButton;

Actuator_PusherY1 := Pusher.PusherY1;
Actuator_PusherY2 := Pusher.PusherY2;


IF((Sensor_SorterEmergencyStop) AND (Sensor_StampEmergencyStop) AND (Sensor_MagazinEmergencyStop))THEN
	Mag();
	Crane();
	Stamp();
	Conveyor();
	Pusher();
	IF((Actuator_SorterGreenLampConveyor) AND (Actuator_MagazinGreenLamp) AND (Actuator_StampGreenLamp))THEN
		IF((Stamp.StartCommandStamp) AND (Crane.StartCommandCrane) AND (Conveyor.StartCommandConveyor) AND (Mag.StartCommandMagazin))THEN
			Crane.StartVar := TRUE;
			Conveyor.StartVar := TRUE;
			Mag.StartVar := TRUE;
			Pusher.StartVar := TRUE;
			Stamp.StartVar := TRUE;
		END_IF
	END_IF
	Crane.SFCReset := FALSE;
	Conveyor.SFCReset := FALSE;
	Mag.SFCReset := FALSE;
	Pusher.SFCReset := FALSE;
	Stamp.SFCReset := FALSE;
ELSIF ((NOT Sensor_SorterEmergencyStop) OR (NOT Sensor_StampEmergencyStop) OR (NOT Sensor_MagazinEmergencyStop))THEN
	Actuator_MagazinSlider := FALSE;
	Actuator_CraneLower := FALSE;
	Actuator_MagazinVacuumOn := FALSE;
	Actuator_MagazinVacuumOff := TRUE;
	Actuator_MagazinGreenLamp := FALSE;
	Actuator_CraneTurnCounterclockwise := FALSE;
	Actuator_CraneTurnClockwise := FALSE;
	Actuator_SorterConveyorTowardsStacker := FALSE;
	Actuator_SorterConveyorTowardsCrane := FALSE;
	Actuator_SorterGreenLampConveyor := FALSE;
	Actuator_PusherY1 := FALSE;
	Actuator_PusherY2 := FALSE;
	Actuator_StampSliderMovedOut := TRUE;
	Actuator_StampSliderMovedIn := FALSE;
	Actuator_StampGreenLamp := FALSE;
	Actuator_StampPusher := FALSE;

	Actuator_AnalogCranePressure := 0;
	
	Crane.SFCReset := TRUE;
	Conveyor.SFCReset := TRUE;
	Mag.SFCReset := TRUE;
	Pusher.SFCReset := TRUE;
	Stamp.SFCReset := TRUE;
	
	Crane.StartVar := FALSE;
	Conveyor.StartVar := FALSE;
	Mag.StartVar := FALSE;
	Pusher.StartVar := FALSE;
	Stamp.StartVar := FALSE;
END_IF

          
END_PROGRAM

FUNCTION_BLOCK Stamp
  VAR_INPUT
    StampSliderSensorMovedOut : BOOL;
    StampSliderSensorMovedIn : BOOL;
    StampSliderFilled : BOOL;
    StampUp : BOOL;
    StampLowered : BOOL;
    CraneDown : BOOL;
    CraneUp : BOOL;
    CraneSucked : BOOL;
    CranePositionStamp : BOOL;
    CraneOnConveyor : BOOL;
    AnalogCranePosition : INT;
    StampStartButton : BOOL;
    SFCReset : BOOL;
    StartVar : BOOL;
  END_VAR
  VAR_OUTPUT
    StampSliderMovedOut : BOOL;
    StampSliderMovedIn : BOOL;
    StampWhiteLamp : BOOL;
    StampPusher : BOOL;
    StampGreenLamp : BOOL;
    StampPressure : BOOL;
    StartCommandStamp : BOOL;
  END_VAR
  VAR
    interconnect : BOOL;
    Timer : TON;
    Duration : TIME := TIME#500ms;
    interconnectStampStartCommand : BOOL;
    SFCInit : BOOL;
  END_VAR

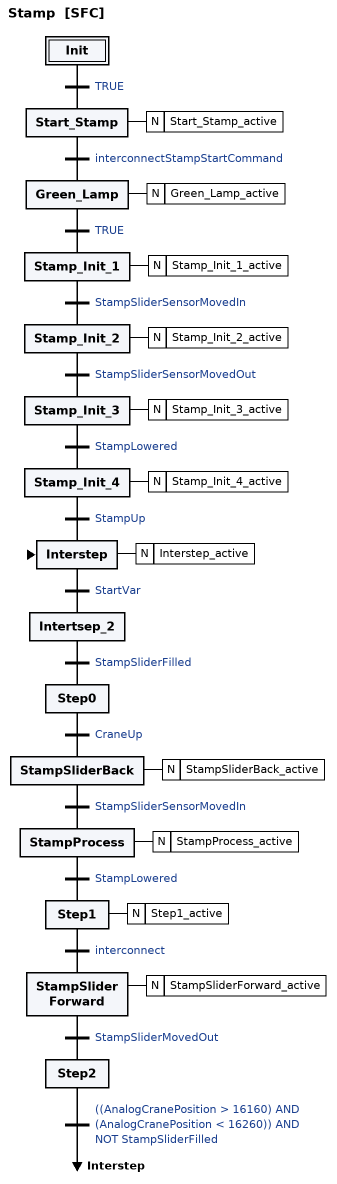
INITIAL_STEP Init:
END_STEP
TRANSITION FROM Init TO Start_Stamp
  := TRUE;
END_TRANSITION
STEP Start_Stamp:
  Start_Stamp_active(N);
END_STEP
TRANSITION FROM Start_Stamp TO Green_Lamp
  := interconnectStampStartCommand;
END_TRANSITION
STEP Green_Lamp:
  Green_Lamp_active(N);
END_STEP
TRANSITION FROM Green_Lamp TO Stamp_Init_1
  := TRUE;
END_TRANSITION
STEP Stamp_Init_1:
  Stamp_Init_1_active(N);
END_STEP
TRANSITION FROM Stamp_Init_1 TO Stamp_Init_2
  := StampSliderSensorMovedIn;
END_TRANSITION
STEP Stamp_Init_2:
  Stamp_Init_2_active(N);
END_STEP
TRANSITION FROM Stamp_Init_2 TO Stamp_Init_3
  := StampSliderSensorMovedOut;
END_TRANSITION
STEP Stamp_Init_3:
  Stamp_Init_3_active(N);
END_STEP
TRANSITION FROM Stamp_Init_3 TO Stamp_Init_4
  := StampLowered;
END_TRANSITION
STEP Stamp_Init_4:
  Stamp_Init_4_active(N);
END_STEP
TRANSITION FROM Stamp_Init_4 TO Interstep
  := StampUp;
END_TRANSITION
STEP Interstep:
  Interstep_active(N);
END_STEP
TRANSITION FROM Interstep TO Intertsep_2
  := StartVar;
END_TRANSITION
STEP Intertsep_2:
END_STEP
TRANSITION FROM Intertsep_2 TO Step0
  := StampSliderFilled;
END_TRANSITION
STEP Step0:
END_STEP
TRANSITION FROM Step0 TO StampSliderBack
  := CraneUp;
END_TRANSITION
STEP StampSliderBack:
  StampSliderBack_active(N);
END_STEP
TRANSITION FROM StampSliderBack TO StampProcess
  := StampSliderSensorMovedIn;
END_TRANSITION
STEP StampProcess:
  StampProcess_active(N);
END_STEP
TRANSITION FROM StampProcess TO Step1
  := StampLowered;
END_TRANSITION
STEP Step1:
  Step1_active(N);
END_STEP
TRANSITION FROM Step1 TO StampSliderForward
  := interconnect;
END_TRANSITION
STEP StampSliderForward:
  StampSliderForward_active(N);
END_STEP
TRANSITION FROM StampSliderForward TO Step2
  := StampSliderMovedOut;
END_TRANSITION
STEP Step2:
END_STEP
TRANSITION FROM Step2 TO Interstep
  := ((AnalogCranePosition > 16160) AND (AnalogCranePosition < 16260)) AND NOT StampSliderFilled;
END_TRANSITION

ACTION Stamp_Init_3_active:
                StampPusher := TRUE;
              
END_ACTION

ACTION StampSliderForward_active:
                StampPusher := FALSE;
StampSliderMovedOut := TRUE;

IF((StampLowered=FALSE)AND(StampUp=TRUE))THEN
	interconnect := FALSE;
END_IF

Timer(IN:=FALSE, PT:=T#1ms);
              
END_ACTION

ACTION StampSliderBack_active:
                StampSliderMovedIn := TRUE;
StampSliderMovedOut := FALSE;
              
END_ACTION

ACTION Stamp_Init_2_active:
                StampSliderMovedIn := FALSE;
StampSliderMovedOut := TRUE;
              
END_ACTION

ACTION Step1_active:
                Timer(IN:=StampLowered, PT:=T#500MS);
interconnect := Timer.Q;
              
END_ACTION

ACTION Interstep_active:
                StartCommandStamp := TRUE;
              
END_ACTION

ACTION Green_Lamp_active:
                StampGreenLamp := TRUE;
interconnectStampStartCommand := FALSE;
              
END_ACTION

ACTION Stamp_Init_1_active:
                StampSliderMovedIn := TRUE;
StampSliderMovedOut := FALSE;
              
END_ACTION

ACTION Start_Stamp_active:
                StampSliderMovedOut := FALSE;
StampSliderMovedIn := FALSE;
StampPusher := FALSE;
StampGreenLamp := FALSE;
StampPressure := FALSE;
StartCommandStamp := FALSE;


IF(StampStartButton = TRUE) THEN
	interconnectStampStartCommand := TRUE;
END_IF
              
END_ACTION

ACTION StampProcess_active:
                StampSliderMovedIn := FALSE;
StampPusher := TRUE;
              
END_ACTION

ACTION Stamp_Init_4_active:
                StampPusher := FALSE;
              
END_ACTION
END_FUNCTION_BLOCK

FUNCTION_BLOCK Pusher
  VAR_INPUT
    SorterLightnesssensorCraneInterfaceInverse : BOOL;
    SorterLightbarrierCraneInterface : BOOL;
    SorterCapacitiveSensorPusher1 : BOOL;
    SorterLightnessSensorPusher1 : BOOL;
    SorterCapacitiveSensorPusher2 : BOOL;
    SorterLightnessSensorPusher2 : BOOL;
    SorterLightnessSensorPusher3 : BOOL;
    SorterPusher1MovedOut : BOOL;
    SorterPusher1MovedIn : BOOL;
    SorterPusher2MovedOut : BOOL;
    SorterPusher2MovedIn : BOOL;
    SorterStartButton : BOOL;
    SFCReset : BOOL;
    StartVar : BOOL;
  END_VAR
  VAR_OUTPUT
    PusherY1 : BOOL;
    PusherY2 : BOOL;
  END_VAR
  VAR
    Timer2 : TON;  (* enum : INT :=0; Timer1: TON; Duration1: TIME := T#300MS; interconnect : BOOL; *)
    Duration2 : TIME := TIME#2s0ms;
    interconnect2 : BOOL;
    Timer3 : TON;
    Duration3 : TIME := TIME#200ms;
    interconnect3 : BOOL;
    Slide1_white : INT := 1;
    Slide1_black : INT := 1;
    Slide1_metal : INT := 1;
    Slide2_white : INT := 1;
    Slide2_black : INT := 1;
    Slide2_metal : INT := 1;
    Slide3_white : INT := 1;
    Slide3_black : INT := 1;
    Slide3_metal : INT := 1;
    Priority_Var_Black : INT := 3;
    Priority_Var_White : INT := 3;
    Priority_Var_Metal : INT := 3;
    Timer_Slide1_Black : TON;
    Duration_Slide1_Black : TIME := TIME#950ms;
    interconnect_Slide1_Black : BOOL;
    Timer_Slide2_Black : TON;
    Duration_Slide2_Black : TIME := TIME#2s0ms;
    interconnect_Slide2_Black : BOOL;
    Timer_Slide1_White : TON;
    Duration_Slide1_White : TIME := TIME#300ms;
    interconnect_Slide1_White : BOOL;
    Timer_Slide2_White : TON;
    Duration_Slide2_White : TIME := TIME#370ms;
    interconnect_Slide2_White : BOOL;
    Timer_Slide1_Metal : TON;
    Duration_Slide1_Metal : TIME := TIME#300ms;
    interconnect_Slide1_Metal : BOOL;
    Timer_Slide2_Metal : TON;
    Duration_Slide2_Metal : TIME := TIME#370ms;
    interconnect_Slide2_Metal : BOOL;
    SFCInit : BOOL;
  END_VAR

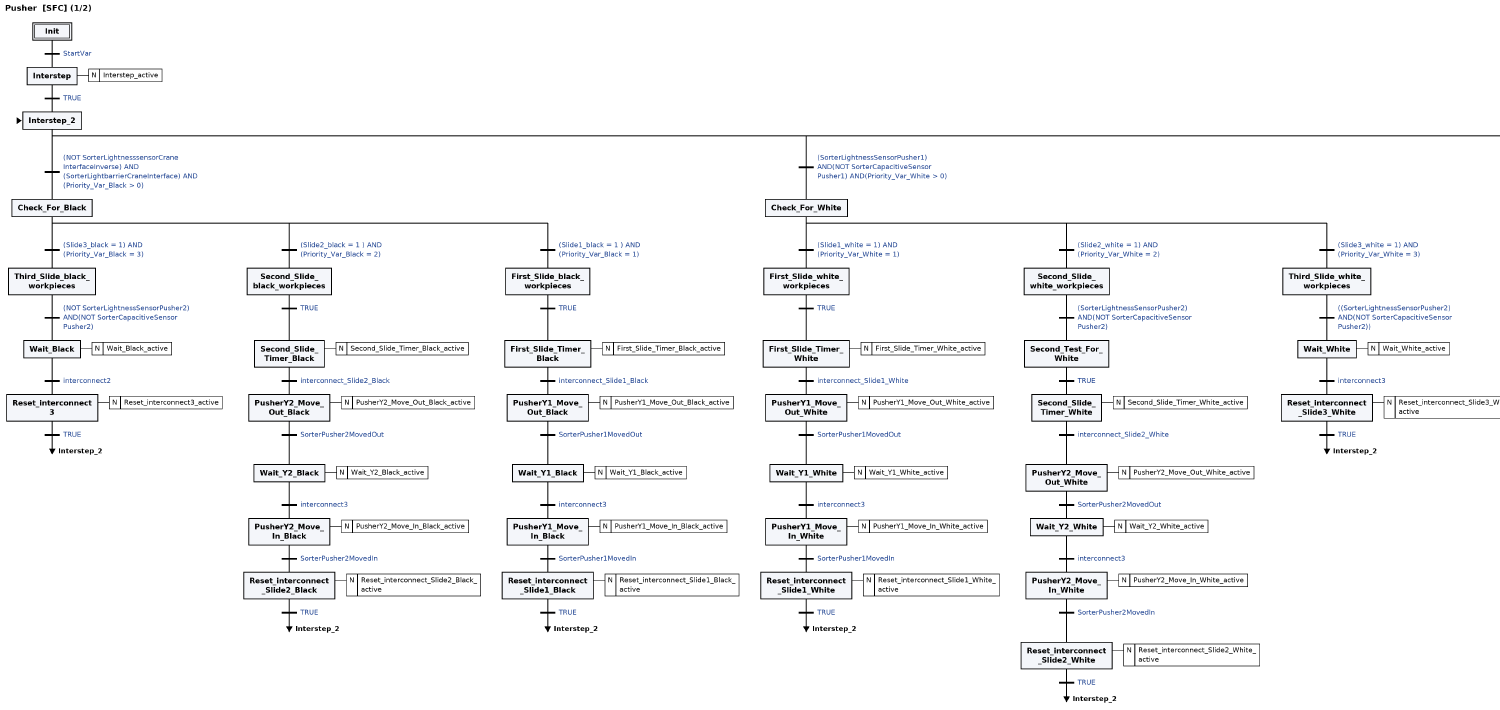
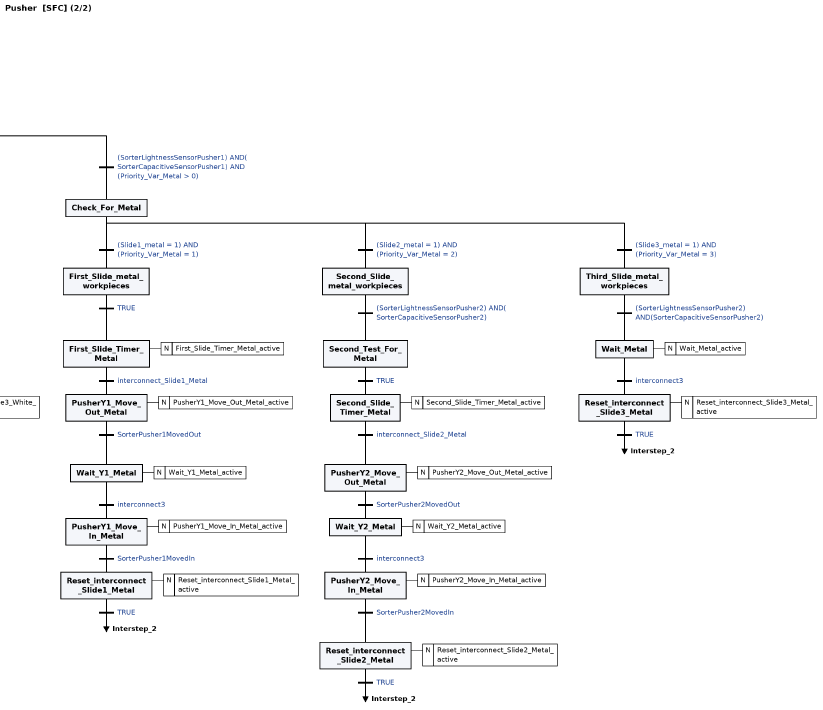
INITIAL_STEP Init:
END_STEP
TRANSITION FROM Init TO Interstep
  := StartVar;
END_TRANSITION
STEP Interstep:
  Interstep_active(N);
END_STEP
TRANSITION FROM Interstep TO Interstep_2
  := TRUE;
END_TRANSITION
STEP Interstep_2:
END_STEP
TRANSITION FROM Interstep_2 TO Check_For_Black
  := (NOT SorterLightnesssensorCraneInterfaceInverse) AND (SorterLightbarrierCraneInterface) AND (Priority_Var_Black > 0);
END_TRANSITION
TRANSITION FROM Interstep_2 TO Check_For_White
  := (SorterLightnessSensorPusher1) AND(NOT SorterCapacitiveSensorPusher1) AND(Priority_Var_White > 0);
END_TRANSITION
TRANSITION FROM Interstep_2 TO Check_For_Metal
  := (SorterLightnessSensorPusher1) AND( SorterCapacitiveSensorPusher1) AND (Priority_Var_Metal > 0);
END_TRANSITION
STEP Check_For_Black:
END_STEP
TRANSITION FROM Check_For_Black TO Third_Slide_black_workpieces
  := (Slide3_black = 1) AND (Priority_Var_Black = 3);
END_TRANSITION
TRANSITION FROM Check_For_Black TO Second_Slide_black_workpieces
  := (Slide2_black = 1 ) AND (Priority_Var_Black = 2);
END_TRANSITION
TRANSITION FROM Check_For_Black TO First_Slide_black_workpieces
  := (Slide1_black = 1 ) AND (Priority_Var_Black = 1);
END_TRANSITION
STEP Third_Slide_black_workpieces:
END_STEP
TRANSITION FROM Third_Slide_black_workpieces TO Wait_Black
  := (NOT SorterLightnessSensorPusher2) AND(NOT SorterCapacitiveSensorPusher2);
END_TRANSITION
STEP Wait_Black:
  Wait_Black_active(N);
END_STEP
TRANSITION FROM Wait_Black TO Reset_interconnect3
  := interconnect2;
END_TRANSITION
STEP Reset_interconnect3:
  Reset_interconnect3_active(N);
END_STEP
TRANSITION FROM Reset_interconnect3 TO Interstep_2
  := TRUE;
END_TRANSITION
STEP Second_Slide_black_workpieces:
END_STEP
TRANSITION FROM Second_Slide_black_workpieces TO Second_Slide_Timer_Black
  := TRUE;
END_TRANSITION
STEP Second_Slide_Timer_Black:
  Second_Slide_Timer_Black_active(N);
END_STEP
TRANSITION FROM Second_Slide_Timer_Black TO PusherY2_Move_Out_Black
  := interconnect_Slide2_Black;
END_TRANSITION
STEP PusherY2_Move_Out_Black:
  PusherY2_Move_Out_Black_active(N);
END_STEP
TRANSITION FROM PusherY2_Move_Out_Black TO Wait_Y2_Black
  := SorterPusher2MovedOut;
END_TRANSITION
STEP Wait_Y2_Black:
  Wait_Y2_Black_active(N);
END_STEP
TRANSITION FROM Wait_Y2_Black TO PusherY2_Move_In_Black
  := interconnect3;
END_TRANSITION
STEP PusherY2_Move_In_Black:
  PusherY2_Move_In_Black_active(N);
END_STEP
TRANSITION FROM PusherY2_Move_In_Black TO Reset_interconnect_Slide2_Black
  := SorterPusher2MovedIn;
END_TRANSITION
STEP Reset_interconnect_Slide2_Black:
  Reset_interconnect_Slide2_Black_active(N);
END_STEP
TRANSITION FROM Reset_interconnect_Slide2_Black TO Interstep_2
  := TRUE;
END_TRANSITION
STEP First_Slide_black_workpieces:
END_STEP
TRANSITION FROM First_Slide_black_workpieces TO First_Slide_Timer_Black
  := TRUE;
END_TRANSITION
STEP First_Slide_Timer_Black:
  First_Slide_Timer_Black_active(N);
END_STEP
TRANSITION FROM First_Slide_Timer_Black TO PusherY1_Move_Out_Black
  := interconnect_Slide1_Black;
END_TRANSITION
STEP PusherY1_Move_Out_Black:
  PusherY1_Move_Out_Black_active(N);
END_STEP
TRANSITION FROM PusherY1_Move_Out_Black TO Wait_Y1_Black
  := SorterPusher1MovedOut;
END_TRANSITION
STEP Wait_Y1_Black:
  Wait_Y1_Black_active(N);
END_STEP
TRANSITION FROM Wait_Y1_Black TO PusherY1_Move_In_Black
  := interconnect3;
END_TRANSITION
STEP PusherY1_Move_In_Black:
  PusherY1_Move_In_Black_active(N);
END_STEP
TRANSITION FROM PusherY1_Move_In_Black TO Reset_interconnect_Slide1_Black
  := SorterPusher1MovedIn;
END_TRANSITION
STEP Reset_interconnect_Slide1_Black:
  Reset_interconnect_Slide1_Black_active(N);
END_STEP
TRANSITION FROM Reset_interconnect_Slide1_Black TO Interstep_2
  := TRUE;
END_TRANSITION
STEP Check_For_White:
END_STEP
TRANSITION FROM Check_For_White TO First_Slide_white_workpieces
  := (Slide1_white = 1) AND (Priority_Var_White = 1);
END_TRANSITION
TRANSITION FROM Check_For_White TO Second_Slide_white_workpieces
  := (Slide2_white = 1) AND (Priority_Var_White = 2);
END_TRANSITION
TRANSITION FROM Check_For_White TO Third_Slide_white_workpieces
  := (Slide3_white = 1) AND (Priority_Var_White = 3);
END_TRANSITION
STEP First_Slide_white_workpieces:
END_STEP
TRANSITION FROM First_Slide_white_workpieces TO First_Slide_Timer_White
  := TRUE;
END_TRANSITION
STEP First_Slide_Timer_White:
  First_Slide_Timer_White_active(N);
END_STEP
TRANSITION FROM First_Slide_Timer_White TO PusherY1_Move_Out_White
  := interconnect_Slide1_White;
END_TRANSITION
STEP PusherY1_Move_Out_White:
  PusherY1_Move_Out_White_active(N);
END_STEP
TRANSITION FROM PusherY1_Move_Out_White TO Wait_Y1_White
  := SorterPusher1MovedOut;
END_TRANSITION
STEP Wait_Y1_White:
  Wait_Y1_White_active(N);
END_STEP
TRANSITION FROM Wait_Y1_White TO PusherY1_Move_In_White
  := interconnect3;
END_TRANSITION
STEP PusherY1_Move_In_White:
  PusherY1_Move_In_White_active(N);
END_STEP
TRANSITION FROM PusherY1_Move_In_White TO Reset_interconnect_Slide1_White
  := SorterPusher1MovedIn;
END_TRANSITION
STEP Reset_interconnect_Slide1_White:
  Reset_interconnect_Slide1_White_active(N);
END_STEP
TRANSITION FROM Reset_interconnect_Slide1_White TO Interstep_2
  := TRUE;
END_TRANSITION
STEP Second_Slide_white_workpieces:
END_STEP
TRANSITION FROM Second_Slide_white_workpieces TO Second_Test_For_White
  := (SorterLightnessSensorPusher2) AND(NOT SorterCapacitiveSensorPusher2);
END_TRANSITION
STEP Second_Test_For_White:
END_STEP
TRANSITION FROM Second_Test_For_White TO Second_Slide_Timer_White
  := TRUE;
END_TRANSITION
STEP Second_Slide_Timer_White:
  Second_Slide_Timer_White_active(N);
END_STEP
TRANSITION FROM Second_Slide_Timer_White TO PusherY2_Move_Out_White
  := interconnect_Slide2_White;
END_TRANSITION
STEP PusherY2_Move_Out_White:
  PusherY2_Move_Out_White_active(N);
END_STEP
TRANSITION FROM PusherY2_Move_Out_White TO Wait_Y2_White
  := SorterPusher2MovedOut;
END_TRANSITION
STEP Wait_Y2_White:
  Wait_Y2_White_active(N);
END_STEP
TRANSITION FROM Wait_Y2_White TO PusherY2_Move_In_White
  := interconnect3;
END_TRANSITION
STEP PusherY2_Move_In_White:
  PusherY2_Move_In_White_active(N);
END_STEP
TRANSITION FROM PusherY2_Move_In_White TO Reset_interconnect_Slide2_White
  := SorterPusher2MovedIn;
END_TRANSITION
STEP Reset_interconnect_Slide2_White:
  Reset_interconnect_Slide2_White_active(N);
END_STEP
TRANSITION FROM Reset_interconnect_Slide2_White TO Interstep_2
  := TRUE;
END_TRANSITION
STEP Third_Slide_white_workpieces:
END_STEP
TRANSITION FROM Third_Slide_white_workpieces TO Wait_White
  := ((SorterLightnessSensorPusher2) AND(NOT SorterCapacitiveSensorPusher2));
END_TRANSITION
STEP Wait_White:
  Wait_White_active(N);
END_STEP
TRANSITION FROM Wait_White TO Reset_interconnect_Slide3_White
  := interconnect3;
END_TRANSITION
STEP Reset_interconnect_Slide3_White:
  Reset_interconnect_Slide3_White_active(N);
END_STEP
TRANSITION FROM Reset_interconnect_Slide3_White TO Interstep_2
  := TRUE;
END_TRANSITION
STEP Check_For_Metal:
END_STEP
TRANSITION FROM Check_For_Metal TO First_Slide_metal_workpieces
  := (Slide1_metal = 1) AND (Priority_Var_Metal = 1);
END_TRANSITION
TRANSITION FROM Check_For_Metal TO Second_Slide_metal_workpieces
  := (Slide2_metal = 1) AND (Priority_Var_Metal = 2);
END_TRANSITION
TRANSITION FROM Check_For_Metal TO Third_Slide_metal_workpieces
  := (Slide3_metal = 1) AND (Priority_Var_Metal = 3);
END_TRANSITION
STEP First_Slide_metal_workpieces:
END_STEP
TRANSITION FROM First_Slide_metal_workpieces TO First_Slide_Timer_Metal
  := TRUE;
END_TRANSITION
STEP First_Slide_Timer_Metal:
  First_Slide_Timer_Metal_active(N);
END_STEP
TRANSITION FROM First_Slide_Timer_Metal TO PusherY1_Move_Out_Metal
  := interconnect_Slide1_Metal;
END_TRANSITION
STEP PusherY1_Move_Out_Metal:
  PusherY1_Move_Out_Metal_active(N);
END_STEP
TRANSITION FROM PusherY1_Move_Out_Metal TO Wait_Y1_Metal
  := SorterPusher1MovedOut;
END_TRANSITION
STEP Wait_Y1_Metal:
  Wait_Y1_Metal_active(N);
END_STEP
TRANSITION FROM Wait_Y1_Metal TO PusherY1_Move_In_Metal
  := interconnect3;
END_TRANSITION
STEP PusherY1_Move_In_Metal:
  PusherY1_Move_In_Metal_active(N);
END_STEP
TRANSITION FROM PusherY1_Move_In_Metal TO Reset_interconnect_Slide1_Metal
  := SorterPusher1MovedIn;
END_TRANSITION
STEP Reset_interconnect_Slide1_Metal:
  Reset_interconnect_Slide1_Metal_active(N);
END_STEP
TRANSITION FROM Reset_interconnect_Slide1_Metal TO Interstep_2
  := TRUE;
END_TRANSITION
STEP Second_Slide_metal_workpieces:
END_STEP
TRANSITION FROM Second_Slide_metal_workpieces TO Second_Test_For_Metal
  := (SorterLightnessSensorPusher2) AND( SorterCapacitiveSensorPusher2);
END_TRANSITION
STEP Second_Test_For_Metal:
END_STEP
TRANSITION FROM Second_Test_For_Metal TO Second_Slide_Timer_Metal
  := TRUE;
END_TRANSITION
STEP Second_Slide_Timer_Metal:
  Second_Slide_Timer_Metal_active(N);
END_STEP
TRANSITION FROM Second_Slide_Timer_Metal TO PusherY2_Move_Out_Metal
  := interconnect_Slide2_Metal;
END_TRANSITION
STEP PusherY2_Move_Out_Metal:
  PusherY2_Move_Out_Metal_active(N);
END_STEP
TRANSITION FROM PusherY2_Move_Out_Metal TO Wait_Y2_Metal
  := SorterPusher2MovedOut;
END_TRANSITION
STEP Wait_Y2_Metal:
  Wait_Y2_Metal_active(N);
END_STEP
TRANSITION FROM Wait_Y2_Metal TO PusherY2_Move_In_Metal
  := interconnect3;
END_TRANSITION
STEP PusherY2_Move_In_Metal:
  PusherY2_Move_In_Metal_active(N);
END_STEP
TRANSITION FROM PusherY2_Move_In_Metal TO Reset_interconnect_Slide2_Metal
  := SorterPusher2MovedIn;
END_TRANSITION
STEP Reset_interconnect_Slide2_Metal:
  Reset_interconnect_Slide2_Metal_active(N);
END_STEP
TRANSITION FROM Reset_interconnect_Slide2_Metal TO Interstep_2
  := TRUE;
END_TRANSITION
STEP Third_Slide_metal_workpieces:
END_STEP
TRANSITION FROM Third_Slide_metal_workpieces TO Wait_Metal
  := (SorterLightnessSensorPusher2) AND(SorterCapacitiveSensorPusher2);
END_TRANSITION
STEP Wait_Metal:
  Wait_Metal_active(N);
END_STEP
TRANSITION FROM Wait_Metal TO Reset_interconnect_Slide3_Metal
  := interconnect3;
END_TRANSITION
STEP Reset_interconnect_Slide3_Metal:
  Reset_interconnect_Slide3_Metal_active(N);
END_STEP
TRANSITION FROM Reset_interconnect_Slide3_Metal TO Interstep_2
  := TRUE;
END_TRANSITION

ACTION PusherY1_Move_Out_Metal_active:
                IF((SorterPusher1MovedOut = FALSE) AND (SorterPusher1MovedIn = TRUE)) THEN
	PusherY1 := TRUE;
END_IF
              
END_ACTION

ACTION Reset_interconnect_Slide1_White_active:
                interconnect3 := FALSE;
Timer3(IN:=FALSE,PT:=T#0MS);
interconnect_Slide1_White := FALSE;
Timer_Slide1_White(IN:=FALSE,PT:=T#0MS);
Slide1_white := Slide1_white - 1;
Priority_Var_White := Priority_Var_White - 1;
              
END_ACTION

ACTION Reset_interconnect_Slide1_Black_active:
                interconnect3 := FALSE;
Timer3(IN:=FALSE,PT:=T#0MS);
interconnect_Slide1_Black := FALSE;
Timer_Slide1_Black(IN:=FALSE,PT:=T#0MS);
Slide1_black := Slide1_black - 1;
Priority_Var_Black := Priority_Var_Black - 1;
              
END_ACTION

ACTION PusherY2_Move_In_Metal_active:
                IF((SorterPusher2MovedOut = TRUE) AND (SorterPusher2MovedIn = FALSE)) THEN
	PusherY2 := FALSE;
END_IF
              
END_ACTION

ACTION Wait_Y1_White_active:
                IF(PusherY1 = TRUE) THEN
	Timer3(IN:=PusherY1, PT:=Duration3);
	interconnect3 := Timer3.Q;
END_IF
              
END_ACTION

ACTION Second_Slide_Timer_White_active:
                Timer_Slide2_White(IN:=TRUE, PT:=Duration_Slide2_White);
interconnect_Slide2_White := Timer_Slide2_White.Q;
              
END_ACTION

ACTION Reset_interconnect_Slide3_White_active:
                interconnect3 := FALSE;
Timer3(IN:=FALSE,PT:=T#0MS);
Slide3_white := Slide3_white - 1;
Priority_Var_White := Priority_Var_White - 1;
              
END_ACTION

ACTION PusherY2_Move_In_White_active:
                IF((SorterPusher2MovedOut = TRUE) AND (SorterPusher2MovedIn = FALSE)) THEN
	PusherY2 := FALSE;
END_IF
              
END_ACTION

ACTION PusherY2_Move_Out_Black_active:
                IF((SorterPusher2MovedOut = FALSE) AND (SorterPusher2MovedIn = TRUE)) THEN
	PusherY2 := TRUE;
END_IF
              
END_ACTION

ACTION PusherY1_Move_In_Metal_active:
                IF((SorterPusher1MovedOut = TRUE) AND (SorterPusher1MovedIn = FALSE)) THEN
	PusherY1 := FALSE;
END_IF
              
END_ACTION

ACTION Wait_Black_active:
                IF(((NOT SorterLightnessSensorPusher2) AND(NOT SorterCapacitiveSensorPusher2)) = TRUE) THEN
	Timer2(IN:=((NOT SorterLightnessSensorPusher2) AND(NOT SorterCapacitiveSensorPusher2)), PT:=Duration2);
	interconnect2 := Timer2.Q;
END_IF
              
END_ACTION

ACTION Wait_White_active:
                Timer3(IN:=TRUE, PT:=Duration3);
	(*Timer3(IN:=((SorterLightnessSensorPusher2) AND(NOT SorterCapacitiveSensorPusher2)), PT:=Duration3);*)
interconnect3 := Timer3.Q;
              
END_ACTION

ACTION PusherY1_Move_Out_Black_active:
                IF((SorterPusher1MovedOut = FALSE) AND (SorterPusher1MovedIn = TRUE)) THEN
	PusherY1 := TRUE;
END_IF
              
END_ACTION

ACTION Second_Slide_Timer_Black_active:
                IF(SorterLightnesssensorCraneInterfaceInverse = TRUE) THEN
	Timer_Slide2_Black(IN:=SorterLightnesssensorCraneInterfaceInverse, PT:=Duration_Slide2_Black);
	interconnect_Slide2_Black := Timer_Slide2_Black.Q;
END_IF
              
END_ACTION

ACTION PusherY2_Move_Out_Metal_active:
                IF((SorterPusher2MovedOut = FALSE) AND (SorterPusher2MovedIn = TRUE)) THEN
	PusherY2 := TRUE;
END_IF
              
END_ACTION

ACTION Reset_interconnect_Slide3_Metal_active:
                interconnect3 := FALSE;
Timer3(IN:=FALSE,PT:=T#0MS);
Slide3_metal := Slide3_metal - 1;
Priority_Var_Metal := Priority_Var_Metal - 1;
              
END_ACTION

ACTION Reset_interconnect_Slide2_Metal_active:
                interconnect3 := FALSE;
Timer3(IN:=FALSE,PT:=T#0MS);
interconnect_Slide2_Metal := FALSE;
Timer_Slide2_Metal(IN:=FALSE,PT:=T#0MS);
Slide2_metal := Slide2_metal - 1;
Priority_Var_Metal := Priority_Var_Metal - 1;
              
END_ACTION

ACTION Wait_Metal_active:
                Timer3(IN:=TRUE, PT:=Duration3);
interconnect3 := Timer3.Q;
              
END_ACTION

ACTION Wait_Y1_Black_active:
                IF(PusherY1 = TRUE) THEN
	Timer3(IN:=PusherY1, PT:=Duration3);
	interconnect3 := Timer3.Q;
END_IF
              
END_ACTION

ACTION Wait_Y1_Metal_active:
                IF(PusherY1 = TRUE) THEN
	Timer3(IN:=PusherY1, PT:=Duration3);
	interconnect3 := Timer3.Q;
END_IF
              
END_ACTION

ACTION PusherY1_Move_In_White_active:
                IF((SorterPusher1MovedOut = TRUE) AND (SorterPusher1MovedIn = FALSE)) THEN
	PusherY1 := FALSE;
END_IF
              
END_ACTION

ACTION Interstep_active:
                PusherY1 := FALSE;
PusherY2 := FALSE;
interconnect2 := FALSE;
interconnect3 := FALSE;
StartVar := FALSE;
interconnect_Slide1_Black := FALSE;
interconnect_Slide2_Black := FALSE;
interconnect_Slide1_White := FALSE;
interconnect_Slide2_White := FALSE;
interconnect_Slide1_Metal := FALSE;
interconnect_Slide2_Metal := FALSE;
              
END_ACTION

ACTION Wait_Y2_Metal_active:
                IF(PusherY2 = TRUE) THEN
	Timer3(IN:=PusherY2, PT:=Duration3);
	interconnect3 := Timer3.Q;
END_IF
              
END_ACTION

ACTION Wait_Y2_White_active:
                IF(PusherY2 = TRUE) THEN
	Timer3(IN:=PusherY2, PT:=Duration3);
	interconnect3 := Timer3.Q;
END_IF
              
END_ACTION

ACTION PusherY2_Move_Out_White_active:
                IF((SorterPusher2MovedOut = FALSE) AND (SorterPusher2MovedIn = TRUE)) THEN
	PusherY2 := TRUE;
END_IF
              
END_ACTION

ACTION First_Slide_Timer_Metal_active:
                Timer_Slide1_Metal(IN:=TRUE, PT:=Duration_Slide1_Metal);
interconnect_Slide1_Metal := Timer_Slide1_Metal.Q;
              
END_ACTION

ACTION Reset_interconnect_Slide1_Metal_active:
                interconnect3 := FALSE;
Timer3(IN:=FALSE,PT:=T#0MS);
interconnect_Slide1_Metal := FALSE;
Timer_Slide1_Metal(IN:=FALSE,PT:=T#0MS);
Slide1_metal := Slide1_metal - 1;
Priority_Var_Metal := Priority_Var_Metal - 1;
              
END_ACTION

ACTION First_Slide_Timer_Black_active:
                IF(SorterLightnesssensorCraneInterfaceInverse = TRUE) THEN
	Timer_Slide1_Black(IN:=SorterLightnesssensorCraneInterfaceInverse, PT:=Duration_Slide1_Black);
	interconnect_Slide1_Black := Timer_Slide1_Black.Q;
END_IF
              
END_ACTION

ACTION Reset_interconnect_Slide2_Black_active:
                interconnect3 := FALSE;
Timer3(IN:=FALSE,PT:=T#0MS);
interconnect_Slide2_Black := FALSE;
Timer_Slide2_Black(IN:=FALSE,PT:=T#0MS);
Slide2_black := Slide2_black - 1;
Priority_Var_Black := Priority_Var_Black - 1; 
              
END_ACTION

ACTION Second_Slide_Timer_Metal_active:
                Timer_Slide2_Metal(IN:=TRUE, PT:=Duration_Slide2_Metal);
interconnect_Slide2_Metal := Timer_Slide2_Metal.Q;
              
END_ACTION

ACTION First_Slide_Timer_White_active:
                Timer_Slide1_White(IN:=TRUE, PT:=Duration_Slide1_White);
interconnect_Slide1_White := Timer_Slide1_White.Q;
              
END_ACTION

ACTION Wait_Y2_Black_active:
                IF(PusherY2 = TRUE) THEN
	Timer3(IN:=PusherY2, PT:=Duration3);
	interconnect3 := Timer3.Q;
END_IF
              
END_ACTION

ACTION Reset_interconnect_Slide2_White_active:
                interconnect3 := FALSE;
Timer3(IN:=FALSE,PT:=T#0MS);
interconnect_Slide2_White := FALSE;
Timer_Slide2_White(IN:=FALSE,PT:=T#0MS);
Slide2_white := Slide2_white - 1;
Priority_Var_White := Priority_Var_White - 1;
              
END_ACTION

ACTION PusherY1_Move_In_Black_active:
                IF((SorterPusher1MovedOut = TRUE) AND (SorterPusher1MovedIn = FALSE)) THEN
	PusherY1 := FALSE;
END_IF
              
END_ACTION

ACTION PusherY2_Move_In_Black_active:
                IF((SorterPusher2MovedOut = TRUE) AND (SorterPusher2MovedIn = FALSE)) THEN
	PusherY2 := FALSE;
END_IF
              
END_ACTION

ACTION PusherY1_Move_Out_White_active:
                IF((SorterPusher1MovedOut = FALSE) AND (SorterPusher1MovedIn = TRUE)) THEN
	PusherY1 := TRUE;
END_IF
              
END_ACTION

ACTION Reset_interconnect3_active:
                interconnect2 := FALSE;
Timer2(IN:=FALSE,PT:=T#0MS);
Slide3_black := Slide3_black - 1;
Priority_Var_Black := Priority_Var_Black - 1; 
              
END_ACTION
END_FUNCTION_BLOCK
